PROGRAM MAIN
VAR
	fbRGBController : FB_RGBController;
	fbBoxLED : FB_BoxLED;
	

END_VAR

fbRGBController();
fbBoxLED();

END_PROGRAM

(* stored: Version 1.1.0.1, ProductVersion 3.1.4024.12
   POU MAIN: Id {2ff7b83e-9d69-4049-8b2d-19c87bd75e82}, SpecialFunc None *)
